// TIA Portal project "LAB3Simu" (V18)

(* hardware
DEVICE "S7-1500/ET200MP station_1"  S7-1500 station
   slot 0: "Rail_0"  Rack  6ES7 590-1***0-0AA0
   slot 1: "PLC_1"  CPU 1511-1 PN  6ES7 511-1AK00-0AB0  V1.8
      slot 3: "CPU display_1"  6ES7591-1AA00-0AA0
      slot 32768: "PROFINET interface_1"  X1
         slot 32769: "Port_1"  X1 P1
         slot 32770: "Port_2"  X1 P2
   slot 2: "CM 1542-5_1"  CM 1542-5  6GK7 542-5DX00-0XE0  V1.0
   slot 3: "DI 16x24VDC HF_1"  DI 16x24VDC HF  6ES7 521-1BH00-0AB0  V1.0
   slot 4: "DQ 16x24VDC/0.5A ST_1"  DQ 16x24VDC/0.5A ST  6ES7 522-1BH00-0AB0  V1.0
   slot 5: "AI 8xU/I/RTD/TC ST_1"  AI 8xU/I/RTD/TC ST  6ES7 531-7KF00-0AB0  V1.0
   slot 6: "AQ 4xU/I ST_1"  AQ 4xU/I ST  6ES7 532-5HD00-0AB0  V1.0
DEVICE "HMI_1"  KTP600 Basic color PN SIPLUS
   slot 0: "HMI_1"  KTP600 Basic color PN SIPLUS  6AG1 647-0AD11-2AX0  12.0.0.0
   slot 1: "HMI_RT_1"  KTP600 Basic color PN SIPLUS  6AG1 647-0AD11-2AX0  12.0.0.0
   slot 5: "HMI_1.IE_CP_1"  PROFINET Interface  12.0.0.0
      slot 1: "PROFINET Interface_1"  PROFINET Interface
         slot 1: "Port_1"  Port
*)

// ===== PLC "PLC_1"  CPU 1511-1 PN =====

VAR_GLOBAL   // PLC tag table "Default tag table"
   "Tag_1" AT %M0.0 : Bool;
   "Tag_2" AT %M0.1 : Bool;
   "Tag_3" AT %M0.2 : Bool;
   "Tag_4" AT %M0.3 : Bool;
   "Tag_5" AT %M0.4 : Bool;
   "Tag_6" AT %M0.5 : Bool;
   "Tag_7" AT %M0.6 : Bool;
   "Start" AT %M1.0 : Bool;
   "Stop" AT %M1.1 : Bool;
   "Emergency" AT %M1.2 : Bool;
   "E_Botellas" AT %M2.0 : Bool;
   "R_Botellas" AT %M2.1 : Bool;
   "Completo_Botellas" AT %M2.2 : Bool;
   "N_Botellas" AT %MW3 : Int;
   "R_Pulsos" AT %M5.0 : Bool;
   "E_Pulsos" AT %M5.1 : Bool;
   "T_Pulsos" AT %MW6 : Int;
   "E_TEstable" AT %M8.0 : Bool;
   "Completo_TEstable" AT %M8.1 : Bool;
   "T_Estable" AT %MD10 : Time;
   "E_Llenado" AT %M14.0 : Bool;
   "Total_Llenado" AT %M14.1 : Bool;
   "T_Llenado" AT %MD15 : Time;
   "Valvula" AT %M20.0 : Bool;
   "Servo_R" AT %M20.1 : Bool;
   "Servo_F" AT %M20.2 : Bool;
   "Servo_E" AT %M20.3 : Bool;
   "Botellas" AT %MW30 : Int;
   "Estado_E" AT %M40.0 : Bool;
   "Estado_S" AT %M40.1 : Bool;
   "Proceso" AT %M40.2 : Bool;
END_VAR

DATA_BLOCK "Generador_DB"   // DB1
{ S7_Optimized_Access := 'TRUE' }
VERSION : 0.1
// stored: InstanceOfName Generador
"Generador"
BEGIN
END_DATA_BLOCK

DATA_BLOCK "Contadores y Temporizadores_DB"   // DB2
{ S7_Optimized_Access := 'TRUE' }
VERSION : 0.1
// stored: InstanceOfName Contadores y Temporizadores
"Contadores y Temporizadores"
BEGIN
END_DATA_BLOCK

DATA_BLOCK "Grafcet_DB"   // DB3
{ S7_Optimized_Access := 'TRUE' }
VERSION : 0.1
// stored: InstanceOfName Grafcet
"Grafcet"
BEGIN
END_DATA_BLOCK

FUNCTION_BLOCK "Generador"   // FB1, STL
{ S7_Optimized_Access := 'TRUE' }
VERSION : 0.1
   VAR
      IEC_Timer_0_Instance : TON_LTIME;
      DB1 : TON_LTIME;
   END_VAR
BEGIN

REGION Network 1
   // Habilitación
         A     "Tag_1";
         =     "Tag_2";

   // Enable T1
         A     "Tag_2";
         AN    "Tag_3";
         =     "Tag_4";

         CALL  #DB1
         ( IN := "Tag_4",
           PT := LT#25000ns,
           Q  := "Tag_5",
           ET :=
         );



   // Enable T2
         A     "Tag_2";
         A     "Tag_5";
         =     "Tag_6";

         CALL  #IEC_Timer_0_Instance
         ( IN := "Tag_6",
           PT := LT#25000ns,
           Q  := "Tag_3",
           ET :=
         );


   // Salida
         A     "Tag_5";
         =     "Tag_7";
END_REGION
END_FUNCTION_BLOCK

FUNCTION_BLOCK "Grafcet"   // FB2, GRAPH_PLUS
{ S7_Optimized_Access := 'TRUE' }
VERSION : 0.1
   VAR_INPUT
      OFF_SQ : Bool := false;   // Turn sequence off
      INIT_SQ : Bool := false;   // Set sequence to initial state
      ACK_EF : Bool := false;   // Acknowledge all errors and faults
      S_PREV : Bool := false;   // Output previous step in parameter S_NO
      S_NEXT : Bool := false;   // Indicate next step in parameter S_NO
      SW_AUTO : Bool := false;   // Automatic mode
      SW_TAP : Bool := false;   // Semiautomatic/switch with transition
      SW_TOP : Bool := false;   // Semiautomatic/ignore transition
      SW_MAN : Bool := false;   // Manual mode
      S_SEL : Int := 0;   // Select step to be output to S_NO
      S_ON : Bool := false;   // Activate step indicated in S_NO
      S_OFF : Bool := false;   // Disable step indicated in S_NO
      T_PUSH : Bool := false;   // Enable transition to switch in semi automatic mode
   END_VAR
   VAR_OUTPUT
      S_NO : Int := 0;   // Step number
      S_MORE : Bool := false;   // More steps are available and can be shown in S_NO
      S_ACTIVE : Bool := false;   // Step indicated in S_NO is active
      ERR_FLT : Bool := false;   // Interlock or supervision group error
      AUTO_ON : Bool := false;   // Automatic mode is active
      TAP_ON : Bool := false;   // Semiautomatic mode/step with transition enabled
      TOP_ON : Bool := false;   // Semiautomatic mode/ignore transition enabled
      MAN_ON : Bool := false;   // Manual mode is active
   END_VAR
   VAR
      HMI_INFO : Array[0..8] of UInt;
      IF_PAR : G7_IfParPlus_V2;
      RT_DATA : G7_RTDataPlus_V2;   // Internal data area
      Trans1 : G7_TransitionPlus_V2;   // Transition structure
      Trans2 : G7_TransitionPlus_V2;   // Transition structure
      Trans3 : G7_TransitionPlus_V2;   // Transition structure
      Trans4 : G7_TransitionPlus_V2;   // Transition structure
      Trans5 : G7_TransitionPlus_V2;   // Transition structure
      Trans6 : G7_TransitionPlus_V2;   // Transition structure
      Trans7 : G7_TransitionPlus_V2;   // Transition structure
      Trans8 : G7_TransitionPlus_V2;   // Transition structure
      Step1 : G7_StepPlus_V2;   // Step structure
      Step2 : G7_StepPlus_V2;   // Step structure
      Step3 : G7_StepPlus_V2;   // Step structure
      Step4 : G7_StepPlus_V2;   // Step structure
      Step5 : G7_StepPlus_V2;   // Step structure
      Step6 : G7_StepPlus_V2;   // Step structure
      Step7 : G7_StepPlus_V2;   // Step structure
      SINI : Array[0..1] of USInt;
      LSTT : Array[0..7] of USInt;
      ATAJ : Array[0..7] of USInt;
      ATAB : Array[0..7] of USInt;
      PSTT : Array[0..7] of USInt;
      NSTT : Array[0..7] of USInt;
      ASSJ : Array[0..6] of USInt;
      ASSB : Array[0..6] of USInt;
      PTTS : Array[0..6] of USInt;
      NTTS : Array[0..6] of USInt;
      SW_SQTS : Array[0..6] of USInt;
      SWITCH : Array[0..1] of USInt;
      TVX : Array[0..3] of USInt;
      TTX : Array[0..3] of USInt;
      TSX : Array[0..1] of USInt;
      S00X : Array[0..1] of USInt;
      SOFFX : Array[0..1] of USInt;
      SONX : Array[0..1] of USInt;
      SAX : Array[0..1] of USInt;
      SERRX : Array[0..7] of USInt;
      SMX : Array[0..7] of USInt;
      S0X : Array[0..7] of USInt;
      S1X : Array[0..7] of USInt;
      IL_ALARM_INST : Program_Alarm;
      SUP_ALARM_INST : Program_Alarm;
      STEP_TIME_ALARM_INST : Program_Alarm;
      IEC_TIMER_INST : IEC_TIMER;
      TRANSACTION_FLAG : Bool := false;
   END_VAR
   // SINI[0] := 2;
   // LSTT[0] := 255;
   // LSTT[1] := 255;
   // LSTT[2] := 255;
   // LSTT[3] := 255;
   // NTTS[4] := 4;
   // ATAJ[1] := 1;
   // ATAJ[2] := 2;
   // ATAJ[3] := 3;
   // PTTS[4] := 3;
   // ASSB[4] := 4;
   // ATAB[1] := 1;
   // ATAB[2] := 2;
   // ATAB[3] := 3;
   // ASSJ[4] := 4;
   // NSTT[4] := 6;
   // PSTT[1] := 1;
   // PSTT[2] := 2;
   // PSTT[3] := 3;
   // PSTT[4] := 4;
   // ATAB[4] := 5;
   // NSTT[0] := 1;
   // NSTT[1] := 2;
   // NSTT[2] := 3;
   // NSTT[3] := 4;
   // ATAJ[4] := 4;
   // LSTT[4] := 255;
   // ASSJ[1] := 1;
   // ASSJ[2] := 2;
   // ASSJ[3] := 3;
   // ASSB[1] := 1;
   // ASSB[2] := 2;
   // ASSB[3] := 3;
   // PTTS[0] := 255;
   // PTTS[2] := 1;
   // PTTS[3] := 2;
   // NTTS[1] := 1;
   // NTTS[2] := 2;
   // NTTS[3] := 3;
   // TVX[0] := 16#1;
   // TTX[0] := 16#1;
   // TSX[0] := 16#1;
   // S00X[0] := 16#1;
   // SOFFX[0] := 16#1;
   // SONX[0] := 16#1;
   // SAX[0] := 16#1;
   // SERRX[0] := 16#1;
   // SMX[0] := 16#1;
   // S0X[0] := 16#1;
   // S1X[0] := 16#1;
   // LSTT[5] := 255;
   // LSTT[6] := 255;
   // ATAJ[5] := 5;
   // ATAJ[6] := 6;
   // ATAB[5] := 4;
   // ATAB[6] := 6;
   // PSTT[5] := 4;
   // PSTT[6] := 5;
   // NSTT[5] := 5;
   // NSTT[6] := 255;
   // ASSJ[5] := 5;
   // ASSB[5] := 5;
   // PTTS[5] := 5;
   // NTTS[5] := 6;
   // SW_SQTS[5] := 1;
   // LSTT[7] := 2;
   // ATAJ[7] := 7;
   // ATAB[7] := 7;
   // PSTT[7] := 6;
   // NSTT[7] := 2;
   // ASSJ[6] := 6;
   // ASSB[6] := 6;
   // PTTS[6] := 4;
   // NTTS[6] := 7;
   // SW_SQTS[6] := 2;
BEGIN
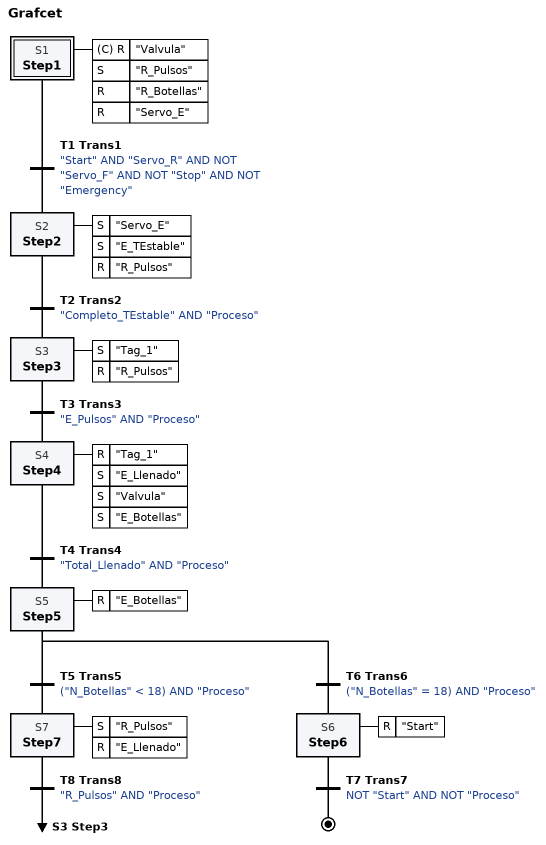
   // sequencer 1
   INITIAL_STEP Step1:   // S1, max time T#10S, warning time T#7S
      (C)     R    "Valvula"
              S    "R_Pulsos"
              R    "R_Botellas"
              R    "Servo_E"
   END_STEP
   TRANSITION Trans1 FROM Step1 TO Step2   // T1
      := "Start" AND "Servo_R" AND NOT "Servo_F" AND NOT "Stop" AND NOT "Emergency";
   END_TRANSITION
   STEP Step2:   // S2, max time T#10S, warning time T#7S
              S    "Servo_E"
              S    "E_TEstable"
              R    "R_Pulsos"
   END_STEP
   TRANSITION Trans2 FROM Step2 TO Step3   // T2
      := "Completo_TEstable" AND "Proceso";
   END_TRANSITION
   STEP Step3:   // S3, max time T#10S, warning time T#7S
              S    "Tag_1"
              R    "R_Pulsos"
   END_STEP
   TRANSITION Trans3 FROM Step3 TO Step4   // T3
      := "E_Pulsos" AND "Proceso";
   END_TRANSITION
   STEP Step5:   // S5, max time T#10S, warning time T#7S
              R    "E_Botellas"
   END_STEP
   TRANSITION Trans5 FROM Step5 TO Step7   // T5
      := ("N_Botellas" < 18) AND "Proceso";
   END_TRANSITION
   TRANSITION Trans6 FROM Step5 TO Step6   // T6
      := ("N_Botellas" = 18) AND "Proceso";
   END_TRANSITION
   STEP Step4:   // S4, max time T#10S, warning time T#7S
              R    "Tag_1"
              S    "E_Llenado"
              S    "Valvula"
              S    "E_Botellas"
   END_STEP
   TRANSITION Trans4 FROM Step4 TO Step5   // T4
      := "Total_Llenado" AND "Proceso";
   END_TRANSITION
   STEP Step6:   // S6, max time T#10S, warning time T#7S
              R    "Start"
   END_STEP
   TRANSITION Trans7 FROM Step6 TO END   // T7
      := NOT "Start" AND NOT "Proceso";
   END_TRANSITION
   STEP Step7:   // S7, max time T#10S, warning time T#7S
              S    "R_Pulsos"
              R    "E_Llenado"
   END_STEP
   TRANSITION Trans8 FROM Step7 TO Step3   // T8, jump
      := "R_Pulsos" AND "Proceso";
   END_TRANSITION
END_FUNCTION_BLOCK

FUNCTION_BLOCK "Contadores y Temporizadores"   // FB3, SCL
{ S7_Optimized_Access := 'TRUE' }
VERSION : 0.1
   VAR RETAIN
      IEC_Counter_0_Instance : CTU_INT;
      IEC_Counter_0_Instance_1 : CTU_INT;
   END_VAR
   VAR
      IEC_Timer_0_Instance : TON_TIME;
      IEC_Timer_0_Instance_1 : TON_TIME;
   END_VAR
BEGIN
   #IEC_Counter_0_Instance(CU := "E_Botellas",
                           R := "R_Botellas",
                           PV := 18,
                           Q => "Completo_Botellas",
                           CV => "N_Botellas");

   #IEC_Counter_0_Instance_1(CU := "Tag_7",
                             R := "R_Pulsos",
                             PV := 500,
                             Q => "E_Pulsos",
                             CV => "T_Pulsos");

   #IEC_Timer_0_Instance(IN := "E_TEstable",
                         PT := T#500ms,
                         Q => "Completo_TEstable",
                         ET => "T_Estable");

   #IEC_Timer_0_Instance_1(IN:="E_Llenado",
                           PT:=T#3s,
                           Q=>"Total_Llenado",
                           ET=>"T_Llenado");
   IF "Start" = 1 THEN
       // Statement section IF
       "Proceso" := TRUE;
       ;
   END_IF;

   IF "Stop" = 1 THEN
       // Statement section IF
       "Proceso" := FALSE;
   ELSE
       "Proceso" := TRUE;
       ;
   END_IF;

   IF "Emergency" = 1 THEN
       // Statement section IF
       "Proceso" := FALSE;
       "R_Botellas" := TRUE;
       "R_Pulsos" := TRUE;
       "Valvula" := FALSE;
       "E_TEstable" := FALSE;
       "E_Llenado" := FALSE;

       ;
   END_IF;
END_FUNCTION_BLOCK

ORGANIZATION_BLOCK "Main"   // OB1, LAD, ProgramCycle
TITLE = "Main Program Sweep (Cycle)"
{ S7_Optimized_Access := 'TRUE' }
VERSION : 0.1
   VAR_INPUT
      Initial_Call : Bool;   // Initial call of this OB
      Remanence : Bool;   // =True, if remanent data are available
   END_VAR
BEGIN

REGION Network 1
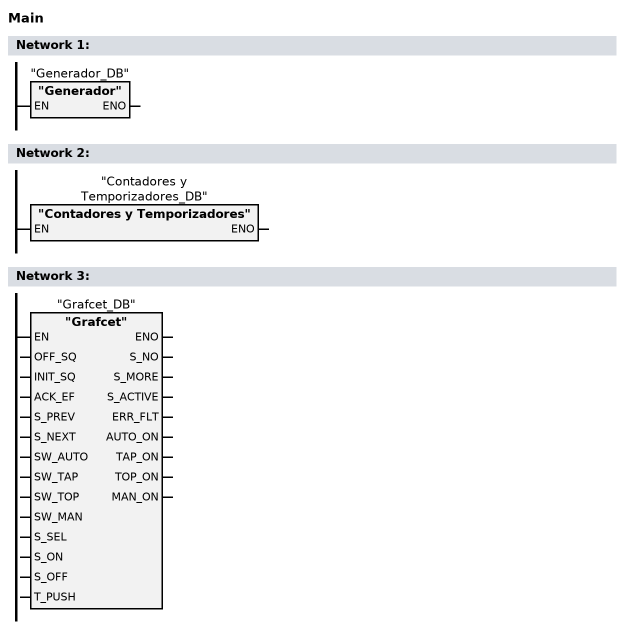
   RUNG wire#powerrail
      "Generador_DB"()
   END_RUNG
   // the same network as SCL:
   "Generador_DB"();   // "Generador"
END_REGION

REGION Network 2
   RUNG wire#powerrail
      "Contadores y Temporizadores_DB"()
   END_RUNG
   // the same network as SCL:
   "Contadores y Temporizadores_DB"();   // "Contadores y Temporizadores"
END_REGION

REGION Network 3
   RUNG wire#powerrail
      "Grafcet_DB"(OFF_SQ :=, INIT_SQ :=, ACK_EF :=, S_PREV :=, S_NEXT :=, SW_AUTO :=, SW_TAP :=, SW_TOP :=, SW_MAN :=, S_SEL :=, S_ON :=, S_OFF :=, T_PUSH :=, S_NO =>, S_MORE =>, S_ACTIVE =>, ERR_FLT =>, AUTO_ON =>, TAP_ON =>, TOP_ON =>, MAN_ON =>)
   END_RUNG
   // the same network as SCL:
   "Grafcet_DB"();   // "Grafcet"
END_REGION
END_ORGANIZATION_BLOCK

(* ===== HMI "HMI_RT_1" =====
system functions are stored by id; their names below are inferred from use
connection "HMI_Connection_1": ETHERNET, SMART_S7_1500_OMS

HMI tags "Default tag table"
   "Tag_ScreenNumber" : UInt, internal
   "Start" : Bool = PLC Start AT %M1.0, 1 s
   "Stop" : Bool = PLC Stop AT %M1.1, 1 s
   "Emergency" : Bool = PLC Emergency AT %M1.2, 1 s

Template "Template_1" 320x240
   Button "Exit" at 266,202 size 52x37; TextOff 'Exit'; PictureOff "ExitRuntime_KTP600_Basic_color_PN"; PictureOn "ExitRuntime_KTP600_Basic_color_PN"
      on Release: StopRuntime(0)
   Button "Template_Button" at 213,202 size 52x37; TextOff 'Text'
   Button "Template_Button_1" at 160,202 size 52x37; TextOff 'Text'
   Button "Template_Button_2" at 107,202 size 52x37; TextOff 'Text'
   Button "Template_Button_3" at 54,202 size 52x37; TextOff 'Text'
   Button "Start screen" at 1,202 size 52x37; TextOff 'Start screen'; PictureOff "NavigateHome_KTP600_Basic_color_PN"; PictureOn "NavigateHome_KTP600_Basic_color_PN"
      on Release: ActivateScreen("Screen_1", 0)
   SymbolicIOField "Symbolic_IO_Field_Screen" at 69,7 size 164x24; TextOff '0'; TextOn '1'; TextList "TextList_ScreenNames"
      ProcessValue <- "Tag_ScreenNumber"
      on Change: ActivateScreenByNumber("Tag_ScreenNumber", 0)
   DateTimeField "HmiScreenItemData" at 235,19 size 85x19
   DateTimeField "HmiScreenItemData_1" at 235,0 size 85x19
   GraphicView "Logo" at 0,0 size 67x38; Picture "Logo of HMI_1"

screen "Screen_1" 320x240
   TextField "Text field_1" at 65,3 size 188x21; Text 'Sistema de Rectificado'
   Circle "Circle_1" at 4,70 size 32x32
      Appearance <- "Start"
   Circle "Circle_2" at 4,114 size 32x32
      Appearance <- "Stop"
   Circle "Circle_3" at 4,160 size 32x32
      Appearance <- "Emergency"
   IOField "I/O field_1" at 214,54 size 96x23
   IOField "I/O field_2" at 214,81 size 96x23
   IOField "I/O field_3" at 214,110 size 96x23
*)